// Block: PPrfArchive1

DATA_BLOCK PPrfArchive1
VERSION : 0.1
   NON_RETAIN
   VAR
      PRG : Array[1..PPRF_TOTAL_ARCHIVE_ITEMS] of PPrf_Data;
   END_VAR

BEGIN
   // No initialization required
END_DATA_BLOCK
